{attribute addProperty BoxType "EP3314-0002-0016"}
{attribute addProperty Id "StatusAT %I*Status_7401E307587.251ValueAT %I*INT16217"}
{attribute addProperty CRC "1130679734"}
{attribute addProperty SizeInBites "74"}
{attribute addProperty SizeInBytes "9.25"}
TYPE TC_TCInputs_Channel_4364CDB6 :
STRUCT
	{attribute addProperty Name "Status"}
	Status AT %I* : Status_7401E307;
	{attribute addProperty Name "Value"}
	Value AT %I* : INT;
END_STRUCT
END_TYPE

(* stored: Version 1.2.0.0, ProductVersion 3.1.4024.9
   DUT TC_TCInputs_Channel_4364CDB6: Id {c3f89019-2679-43f3-af19-f6d2a4e43c8c} *)
